PROGRAM prg_KantoorVerlichting
VAR
	bSchakelaar_1		AT		%I*		:BOOL;
	bSchakelaar_2		AT		%I*		:BOOL;
	bSchakelaar_3		AT		%I*		:BOOL;
	bVerlichting	 	AT 		%Q* 	:BOOL;

	LichtVerlengen: TON;
	TimerVerlichting: TP;
	Flikkeraan: TON;
	FlikkerUit: TOF;
	Flikker: REAL;
	Uitklik: F_TRIG;
	bVerlichtingRaw: BOOL;
END_VAR

LichtVerlengen(IN:= bSchakelaar_1, PT:= T#2S);
TimerVerlichting(IN:= bSchakelaar_1 OR LichtVerlengen.Q, PT:= T#60S, Q=> bVerlichting);

IF TIME_TO_REAL(TimerVerlichting.ET) >= 30 AND Flikker < 3 THEN
	Flikkeraan(IN:= NOT(FlikkerUit.Q) , PT:= T#500MS, Q=> bVerlichting);
	FlikkerUit(IN:= Flikkeraan.Q, PT:= T#500MS);
	Flikker := Flikker+1;
END_IF

IF FlikkerUit.Q THEN
	bVerlichting:=NOT(TimerVerlichting.Q);
ELSE
	bVerlichting:=TimerVerlichting.Q;
END_IF

Uitklik(CLK:= bSchakelaar_1);

IF TIME_TO_REAL(TimerVerlichting.ET) >= 30 AND LichtVerlengen.Q THEN
	TimerVerlichting.IN:=TRUE;
ELSIF bVerlichting AND Uitklik.Q AND NOT(LichtVerlengen.Q) THEN
	bVerlichting:=FALSE;
	TimerVerlichting.IN:=FALSE;
END_IF

END_PROGRAM

(* stored: Version 1.1.0.1, ProductVersion 3.1.4024.15
   POU prg_KantoorVerlichting: Id {b31bbaab-da33-444b-860c-e46c7b080048}, SpecialFunc None *)
